(*
SPDX-FileCopyrightText: © 2026 Oleksandr Tiutyk <trofimich@gmail.com>
SPDX-License-Identifier: MIT
License: https://opensource.org/license/mit
*)

INTERFACE IDemoException EXTENDS TOF_Core.IGeneralException

{attribute 'monitoring' := 'call'}
PROPERTY IsCritical : BOOL
GET
END_GET
END_PROPERTY

METHOD Throw
VAR_INPUT
	sourceNamespaceName : STRING;
	sourceClassName : STRING;
	sourcePOUName : STRING;
	sourcePosition : STRING;
	isCritical : BOOL;
END_VAR
VAR_IN_OUT CONSTANT
	message : STRING(255);
END_VAR
END_METHOD

END_INTERFACE

(* stored: Version 1.1.0.1
   Itf IDemoException: Id {3b6bcc1e-844a-4801-b5aa-14f44145c670}
   Property IsCritical: Id {9cb0087e-b719-46f8-ad18-233c138e2178}
   Get Get: Id {89f67bbf-b032-4415-b7d3-e314a031bf6e}
   Method Throw: Id {2d5d0956-50b1-45bb-94a8-296fb3072af7} *)
